Fanuc KAREL source: KC00022.KL

PROGRAM KC00022
%NOLOCKGROUP
%ENVIRONMENT FLBT
VAR
  I: INTEGER
  J: INTEGER
  K: INTEGER
  R: REAL
  B: BOOLEAN
  S: STRING[80]
  T: STRING[80]
  P: PATH
  Q: PATH
  AI: ARRAY[8] OF INTEGER
  AB: ARRAY[244] OF BYTE
BEGIN
  S = '127.0.0.1'
  MSG_PING(S,I)
END KC00022
